FUNCTION_BLOCK UPDATE (* Event-issuing push button *)
  (* Standard: 61499-2 *)
  (* Version 0.1, 2002-05-03, JHC, Rockwell Automation, Made QI IV=true. *)
  (* Version 0.0, 2001-03-04, JHC, Rockwell Automation, Updated documentation. *)
  (* Compiler header: package fb.rt.hmi; import java.awt.*; import java.awt.event.*; *)
  (* Compiler classdef: public class IN_EVENT extends FBInstance implements ActionListener *)
  (* Compiler Java IBM VisualAge 3.0 *)
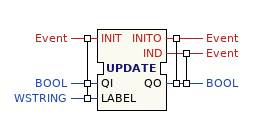
  EVENT_INPUT
    INIT WITH QI, LABEL; (* Service Initialization *)
  END_EVENT
  EVENT_OUTPUT
    INITO WITH QO; (* Initialization Confirm *)
    IND WITH QO; (* Event Indication *)
  END_EVENT
  VAR_INPUT
    QI : BOOL := true;
    LABEL : WSTRING; (* Label *)
  END_VAR
  VAR_OUTPUT
    QO : BOOL;
  END_VAR
  SERVICE FB_BUTTON/Button
    SEQUENCE normal_establishment
      FB_BUTTON.INIT+(LABEL) -> Button.setLabel(LABEL) -> FB_BUTTON.INITO+();
    END_SEQUENCE
    SEQUENCE normal_termination
      FB_BUTTON.INIT-() -> FB_BUTTON.INITO-();
    END_SEQUENCE
    SEQUENCE normal_operation
      Button.actionPerformed(QI=1) -> FB_BUTTON.IND+();
    END_SEQUENCE
    SEQUENCE operation_inhibited
      Button.actionPerformed(QI=0);
    END_SEQUENCE
  END_SERVICE
END_FUNCTION_BLOCK
